FUNCTION_BLOCK FB_Encoder_depth
VAR_INPUT
	Count:REAL;
	mm_per_count:REAL;
	Rope_capping_mode:BOOL;
	Calibrate:BOOL;
	Cal_switch_depth:REAL;
	Cal_window_up:REAL;
	Cal_window_down:REAL;
	Manual_cal:BOOL;
	Manual_cal_depth:REAL;
	Roll_over_count:REAL;
	Reset_offset:BOOL;
	Speed_ave_intervals:REAL;
	Scans_per_update:REAL;
	Brakes_proved_on:BOOL;
	Winder_reset:BOOL;
	Min_depth:REAL;
	Max_depth:REAL;
	Wind_top_depth:REAL;
	Wind_bottom_depth:REAL;
	Mid_wind_error:REAL;
	Direction_hysteresis:REAL;
	Movement_detect_dist:REAL;
END_VAR
VAR_OUTPUT
	Raw_depth:REAL;
	Calibrated_depth:REAL;
	Compensated_depth:REAL;
	Offset:REAL;
	Speed:REAL;
	New_depth:BOOL;
	Going_up:BOOL;
	Movement_detect:BOOL;
	Depth_out_of_range:BOOL;
	Offset_out_of_range:BOOL;
	Closed_above:BOOL;
	Open_below:BOOL;
	Raw_count:REAL;
	Corrected_count:REAL;
END_VAR
VAR_IN_OUT
	hmi_data:dut_hmi_Depth;
	Zero_count:REAL;
	Depth_history:ANY_ARRAY_REAL;
END_VAR
VAR
	Encoder_mm:REAL;
	Captured_depth:REAL;
	Disallow_multiple_cal:BOOL;
	Raw_depth_prev:REAL;
	Scan_count:REAL;
	Late_depth:BOOL;
	Brakes_on_depth:REAL;
	Brakes_proved_on_500ms:BOOL;
	Compensation:REAL;
	Max_pos_reached:REAL;
	hmi_Manual_cal:BOOL;
	Zero_depth_count:REAL;
	FB_WORD_TO_BIT_V0_0: FB_WORD_TO_BIT_V0;
	R_TRIG_0: R_TRIG;
	R_TRIG_1: R_TRIG;
	F_TRIG_0: F_TRIG;
END_VAR

HMI_command();
Corrected_count_m();
Encoder_depth();
Layering_compensation();
Encoder_cal();
Depth_history_m();
Speed_m();
Movement_detect_m();
Direction();
HMI_data_m();

METHOD Corrected_count_m
VAR_INPUT
END_VAR
{warning "TODO: THe last two FB's in this method seem incomplete - no output!}
VAR_INST // added by the converter: edge detectors and wires of the graphical bodies
    _w1, _w2 : REAL;
    _w3 : BOOL;
END_VAR
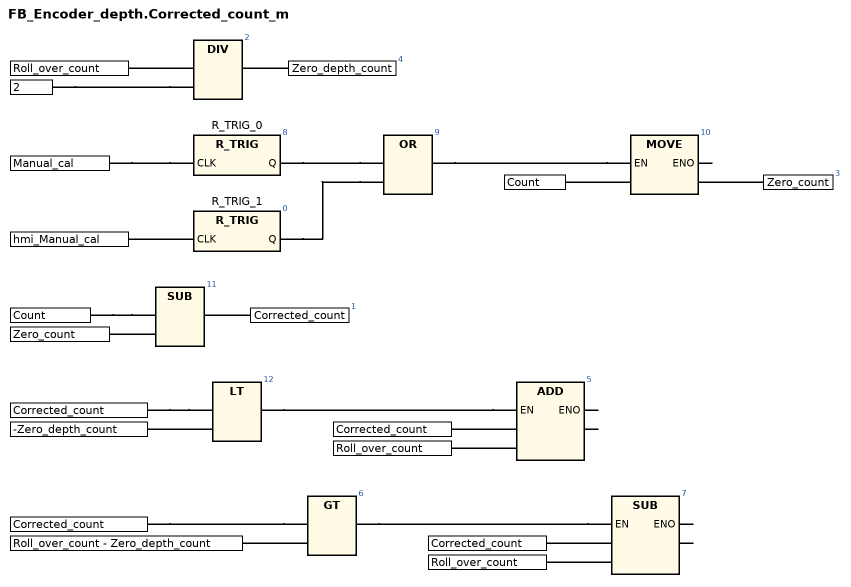
R_TRIG_1(CLK := hmi_Manual_cal); // R_TRIG
Corrected_count := _w1;
Zero_count := _w2;
Zero_depth_count := Roll_over_count / 2;
IF _w3 THEN (* Corrected_count + Roll_over_count; result not used *) END_IF
IF Corrected_count > (Roll_over_count - Zero_depth_count) THEN (* Corrected_count - Roll_over_count; result not used *) END_IF
R_TRIG_0(CLK := Manual_cal); // R_TRIG
IF R_TRIG_0.Q OR R_TRIG_1.Q THEN _w2 := Count; END_IF
_w1 := Count - Zero_count;
_w3 := Corrected_count < (-Zero_depth_count);
END_METHOD

METHOD Encoder_cal
VAR_INPUT
END_VAR
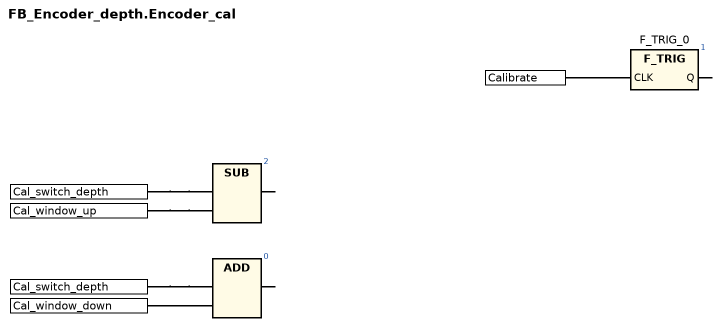
(* Cal_switch_depth + Cal_window_down; result not used *)
F_TRIG_0(CLK := Calibrate); // F_TRIG
(* Cal_switch_depth - Cal_window_up; result not used *)
END_METHOD

METHOD Encoder_depth
VAR_INPUT
END_VAR
VAR_INST // added by the converter: edge detectors and wires of the graphical bodies
    _w1, _w2, _w4 : BOOL;
    _w3, _w6, _w7 : REAL;
    _w5 : ANY;
END_VAR
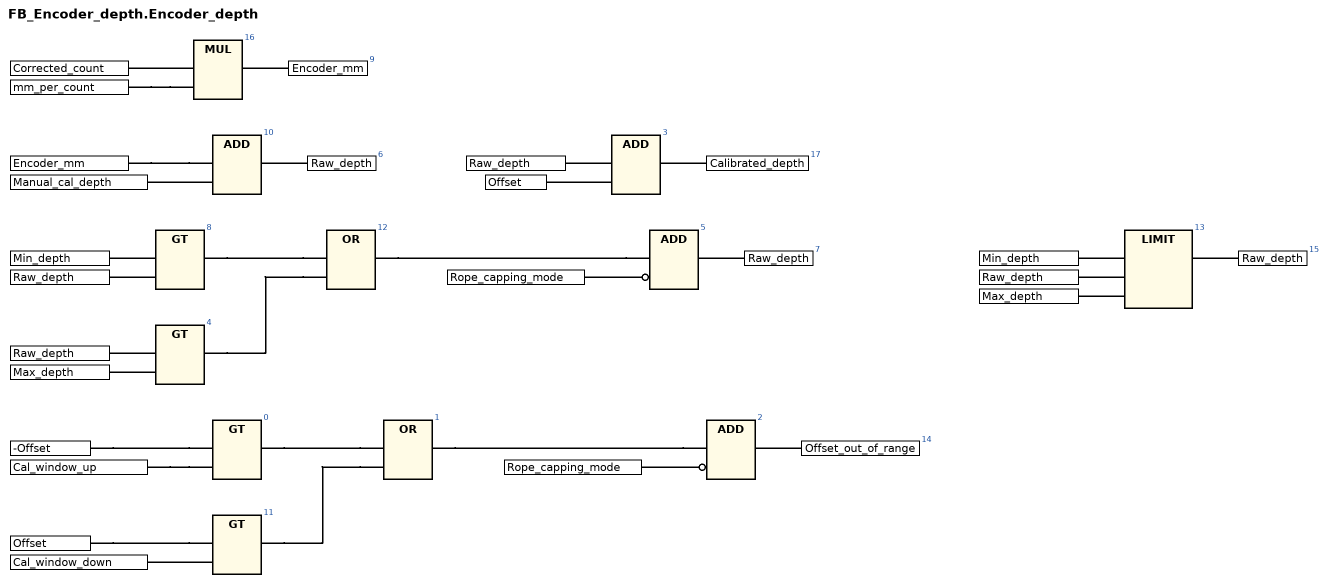
_w2 := ((-Offset) > Cal_window_up OR _w1) + NOT Rope_capping_mode;
_w3 := Raw_depth + Offset;
_w4 := Raw_depth > Max_depth;
Raw_depth := _w6;
Raw_depth := _w5 + NOT Rope_capping_mode;
Encoder_mm := _w7;
_w6 := Encoder_mm + Manual_cal_depth;
_w1 := Offset > Cal_window_down;
_w5 := Min_depth > Raw_depth OR _w4;
Offset_out_of_range := _w2;
Raw_depth := LIMIT(Min_depth, Raw_depth, Max_depth);
_w7 := Corrected_count * mm_per_count;
Calibrated_depth := _w3;
END_METHOD

METHOD HMI_command
VAR_INPUT
END_VAR
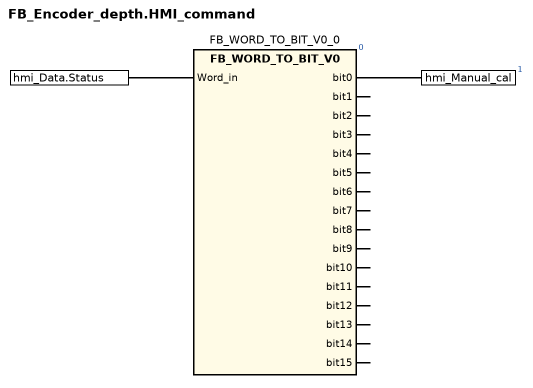
FB_WORD_TO_BIT_V0_0(Word_in := hmi_Data.Status); // FB_WORD_TO_BIT_V0
hmi_Manual_cal := FB_WORD_TO_BIT_V0_0.bit0;
END_METHOD

METHOD Layering_compensation
VAR_INPUT
END_VAR
VAR_INST // added by the converter: edge detectors and wires of the graphical bodies
    _w1 : REAL;
    _w2 : ANY;
END_VAR
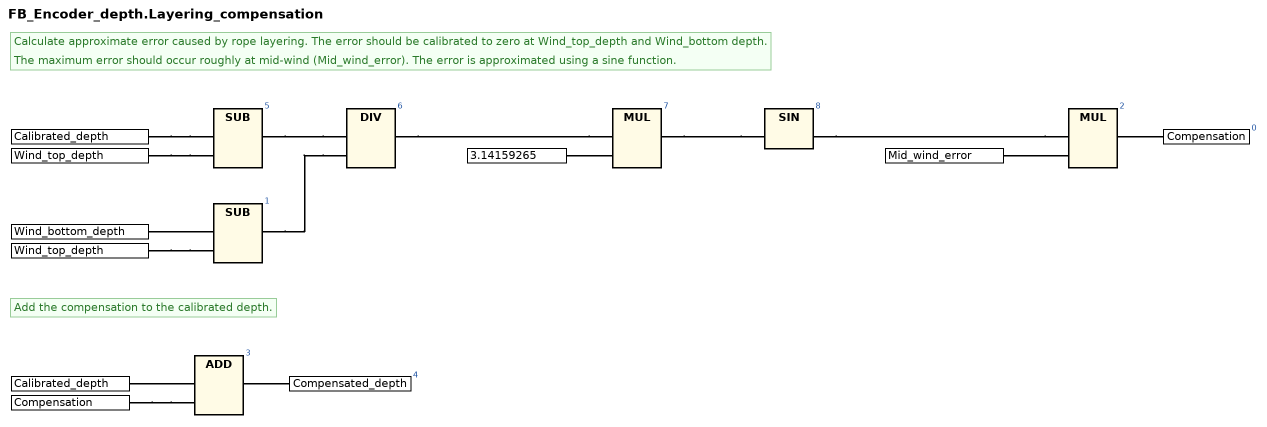
Compensation := _w1;
_w1 := _w2 * Mid_wind_error;
// Add the compensation to the calibrated depth.
Compensated_depth := Calibrated_depth + Compensation;
// Calculate approximate error caused by rope layering. The error should be calibrated to zero at Wind_top_depth and Wind_bottom depth.
// The maximum error should occur roughly at mid-wind (Mid_wind_error). The error is approximated using a sine function.
_w2 := SIN(((Calibrated_depth - Wind_top_depth) / (Wind_bottom_depth - Wind_top_depth)) * 3.14159265);
END_METHOD

END_FUNCTION_BLOCK

(* stored: Version 1.1.0.1, ProductVersion 3.1.4024.0
   POU FB_Encoder_depth: Id {4c58a862-6f56-4a88-80e1-a2ee6717fb65}, SpecialFunc None
   Method Corrected_count_m: Id {ed5f0845-1ee6-4c3d-a20b-d2b00f7d4163}
   Method Encoder_cal: Id {0710b182-8b60-4dc6-b721-2efca8cb3ee8}
   Method Encoder_depth: Id {cd9d7d49-7cce-4412-85d3-0f5676120ee5}
   Method HMI_command: Id {f7f79e77-c5db-40a4-8042-8f519b74941f}
   Method Layering_compensation: Id {1f5bc352-1b4e-4276-a2c2-9276d53f3259} *)
